INTERFACE I_AxisStatus EXTENDS I_StatusEx

METHOD AxisEnabled : BOOL
END_METHOD

PROPERTY AxisID : UDINT
GET
END_GET
END_PROPERTY

PROPERTY AxisState : MC_AxisStates
GET
END_GET
END_PROPERTY

PROPERTY MeasuredAcceleration : LREAL
GET
END_GET
END_PROPERTY

PROPERTY MeasuredPosition : LREAL
GET
END_GET
END_PROPERTY

PROPERTY MeasuredPositionDiff : LREAL
GET
END_GET
END_PROPERTY

PROPERTY MeasuredVelocity : LREAL
GET
END_GET
END_PROPERTY

PROPERTY NegativeMotionIsEnabled : BOOL
GET
END_GET
END_PROPERTY

PROPERTY PositiveMotionIsEnabled : BOOL
GET
END_GET
END_PROPERTY

PROPERTY StandStill : BOOL
GET
END_GET
END_PROPERTY

END_INTERFACE

(* stored: Version 1.1.0.1
   Itf I_AxisStatus: Id {ced1141c-4936-4e2b-89cc-52f3e59358c7}
   Method AxisEnabled: Id {630e5032-35fd-49af-8171-ae8c288f92dd}
   Property AxisID: Id {6a98b3ff-e49f-4c85-a391-34f0ab3ea669}
   Get Get: Id {73635cf1-f38d-42c4-8ee7-552213d89b40}
   Property AxisState: Id {d006c001-4910-47fa-9592-d882dbdfec33}
   Get Get: Id {d4cb8dfa-bc5b-4c9e-b4db-6f401adbeadc}
   Property MeasuredAcceleration: Id {11db257d-9669-4636-bf1c-bca0c2ae5dde}
   Get Get: Id {f4db0f9e-f6fa-470b-a8a6-0964abbcda80}
   Property MeasuredPosition: Id {7e347d7e-a13f-432c-8f4f-b4d6b1f80b41}
   Get Get: Id {bb7cc060-e943-42a2-8ed7-f9b6b4eefec7}
   Property MeasuredPositionDiff: Id {1189e7b1-8db0-42b0-a7e4-fcf97b49effd}
   Get Get: Id {af78f313-84ab-4c3f-8f81-0d297d6cc5b1}
   Property MeasuredVelocity: Id {5404c74a-55c1-4a47-bf7c-750011aa4320}
   Get Get: Id {ecc13acb-39df-4fbd-b1cf-135093881313}
   Property NegativeMotionIsEnabled: Id {2a8dcab0-8683-4ee7-a875-14cdbc960abd}
   Get Get: Id {459b9be0-acd2-465d-b063-5781021bd02f}
   Property PositiveMotionIsEnabled: Id {1411935e-69f0-45ec-be43-8e3a095c1410}
   Get Get: Id {448ecc5b-d498-47b6-9cd0-692c6c199d65}
   Property StandStill: Id {56f881a0-102f-43c3-a476-aa30cefe31e9}
   Get Get: Id {4d5f8519-3e3d-411b-bc51-16b647124219} *)
